// TIA Portal V21 export
TYPE "Std_Segnale"
   STRUCT
      In : Struct
         Segnale : Bool;
      END_STRUCT;
      Prm : Struct
         AbilitaScadenzaForzatura : Bool;
         TempoScadenzaForzatura : "Std_stTimer";
      END_STRUCT;
      Hmi : Struct
         ForzaturaOn : Bool;
         ForzaturaOff : Bool;
         Stato : Int;
      END_STRUCT;
      Out : Struct
         Segnale : Bool;
      END_STRUCT;
   END_STRUCT;
END_TYPE
